FUNCTION_BLOCK SupplyCtrl (* Template for an empty basic function block *)
  (* Standard: 61499-2 *)
  (* Version 1.0, 2018-07-17, az *)
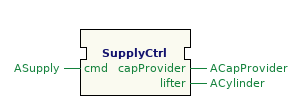
  SOCKETS
    cmd : ASupply;
  END_SOCKETS
  PLUGS
    capProvider : ACapProvider;
    lifter : ACylinder;
  END_PLUGS
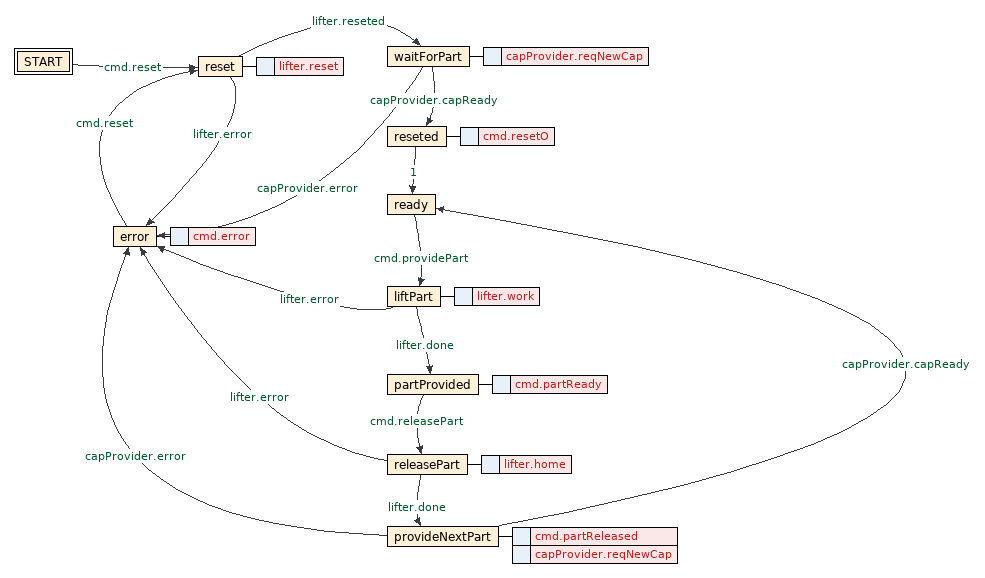
  EC_STATES
    START; (* Initial State *)
    reset : -> lifter.reset;
    error : -> cmd.error;
    waitForPart : -> capProvider.reqNewCap;
    reseted : -> cmd.resetO;
    ready;
    liftPart : -> lifter.work;
    releasePart : -> lifter.home;
    partProvided : -> cmd.partReady;
    provideNextPart : -> cmd.partReleased, -> capProvider.reqNewCap;
  END_STATES
  EC_TRANSITIONS
    START TO reset := cmd.reset;
    error TO reset := cmd.reset;
    reset TO waitForPart := lifter.reseted;
    waitForPart TO reseted := capProvider.capReady;
    reseted TO ready := 1;
    reset TO error := lifter.error;
    ready TO liftPart := cmd.providePart;
    liftPart TO error := lifter.error;
    liftPart TO partProvided := lifter.done;
    partProvided TO releasePart := cmd.releasePart;
    releasePart TO error := lifter.error;
    releasePart TO provideNextPart := lifter.done;
    provideNextPart TO ready := capProvider.capReady;
    waitForPart TO error := capProvider.error;
    provideNextPart TO error := capProvider.error;
  END_TRANSITIONS
END_FUNCTION_BLOCK
